	                #sFB_MCOConveyLinxAixController210(iUDT_AixConfig := #iUDT_Configuration."210".MCO_M01,
	                                                   iUDT_AixInputsModule := #iUDT_MotorInput210,
	                                                   ix_24vOk := #ix_24vOk,
	                                                   ix_SimulationModeActive := "DB_Memory".Simulation,
	                                                   ii_MotorPositionId := 1,
	                                                   qUDT_HMIStatus => #iqUDT_WorkstationStatus."210".MCO_M01,
	                                                   iqUDT_AixOutputsModule := #qUDT_MotorOutput210,
	                                                   iqUDT_ConveyorInterface := #sUDT_Interface210,
	                                                   iqUDT_MCOStatistics := #iqUDT_WorkstationStatistics."210".MCO_M01);
	            END_REGION
	        END_REGION

	        REGION 220

	            REGION Displacement
	                #sFB_Displacement220(#sUDT_Interface220);
	            END_REGION

	            REGION MCO

	                #sFB_MCOConveyLinxAixController220(iUDT_AixConfig := #iUDT_Configuration."220".MCO_M01,
	                                                   iUDT_AixInputsModule := #iUDT_MotorInput220,
	                                                   ix_24vOk := #ix_24vOk,
	                                                   ix_SimulationModeActive := "DB_Memory".Simulation,
	                                                   ii_MotorPositionId := 1,
	                                                   qUDT_HMIStatus => #iqUDT_WorkstationStatus."220".MCO_M01,
	                                                   iqUDT_AixOutputsModule := #qUDT_MotorOutput220,
	                                                   iqUDT_ConveyorInterface := #sUDT_Interface220,
	                                                   iqUDT_MCOStatistics := #iqUDT_WorkstationStatistics."220".MCO_M01);
	            END_REGION
	        END_REGION

	        REGION 221

	            REGION Displacement
	                #sFB_Displacement221(#sUDT_Interface221);
	            END_REGION

	            REGION RAT


	                #sFB_RightAngledTransfer221(iUDT_Configuration := #iUDT_Configuration."221".RightAngledTransfer,
	                                            iUDT_LowerConveyorConfiguration := #iUDT_Configuration."220".Conveyor,
	                                            iUDT_UpperConveyorConfiguration := #iUDT_Configuration."221".Conveyor,
	                                            iUDT_PECConfiguration := #iUDT_Configuration."220".PEC_EoS,
	                                            ii_DestinationA := 0,
	                                            ii_DestinationB := 0,
	                                            ii_DestinationC := 1,
	                                            ii_DestinationD := 0,
	                                            ix_HardwareOk := #ix_HardwareOk,
	                                            ix_400vOk := #ix_400vOk,
	                                            ix_24vOk := #ix_24vOk,
	                                            ix_SafetyOk := #ix_SafetyOk,
	                                            ix_AirPressureOk := #ix_AirPressureOk,
	                                            ix_SectionIsDown := #ix_SectionIsDown221,
	                                            ix_SectionIsUp := #ix_SectionIsUp221,
	                                            ix_ConveyorAAuto := FALSE,
	                                            ix_ConveyorBAuto := #iqUDT_WorkstationCommonStatus."230".AutoON,
	                                            ix_ConveyorCAuto := #iqUDT_WorkstationCommonStatus."210".AutoON,
	                                            ix_ConveyorDAuto := false,
	                                            ix_PEC := #iUDT_MotorInput220.AllSensorPortInputs.LeftSensor,
	                                            ix_ExternalReceiveRequestA := FALSE,
	                                            ix_ExternalReceiveRequestB := FALSE,
	                                            ix_ExternalReceiveRequestC := NOT #iqUDT_WorkstationStatus."210".PEC_EoS.PEC,
	                                            ix_ExternalReceiveRequestD := FALSE,
	                                            ix_PECInfeedC := #iqUDT_WorkstationStatus."210".PEC_EoS.PEC,
	                                            qUDT_HMIRATStatus => #iqUDT_WorkstationStatus."221".RightAngledTransfer,
	                                            qUDT_HMIConveyorStatus => #iqUDT_WorkstationStatus."220".Conveyor,
	                                            qUDT_HMIPECStatus => #iqUDT_WorkstationStatus."221".PEC_EoS,
	                                            qUDT_RATStatus => #iqUDT_WorkstationCommonStatus."221",
	                                            qUDT_ConveyorStatus => #iqUDT_WorkstationCommonStatus."220",
	                                            qx_PopupControl => #qx_PopupControl221,
	                                            qx_ExternalSendRequestA => #tx_dummy,
	                                            qx_ExternalSendRequestB => #tx_dummy,
	                                            qx_ExternalSendRequestC => #tx_dummy,
	                                            qx_ExternalSendRequestD => #tx_dummy,
	                                            iqUDT_EquipmentControl := #iqUDT_EquipmentControl,
	                                            iqUDT_RATCommand := #iqUDT_WorkstationCommands."221".RightAngledTransfer,
	                                            iqUDT_ConveyorCommand := #iqUDT_WorkstationCommands."220".Conveyor,
	                                            iqUDT_RATStatistics := #iqUDT_WorkstationStatistics."221".RightAngledTransfer,
	                                            iqUDT_ConveyorStatistics := #iqUDT_WorkstationStatistics."220".Conveyor,
	                                            iqUDT_PECStatistics := #iqUDT_WorkstationStatistics."221".PEC_EoS,
	                                            iqUDT_HandShakeConveyorA := #tUDT_dummyHandshake,
	                                            iqUDT_HandShakeConveyorB := #sUDT_Handshake220,
	                                            iqUDT_HandShakeConveyorC := #sUDT_Handshake210,
	                                            iqUDT_HandShakeConveyorD := #tUDT_dummyHandshake,
	                                            iqUDT_LowerConveyorInterface := #sUDT_Interface220,
	                                            iqUDT_UpperConveyorInterface := #sUDT_Interface221,
	                                            iqUDT_RATPositioning := #iqUDT_RATPositioning220,
	                                            iqUDT_BladeStopEoSInterface := #tUDT_DummyBladeStop,
	                                            iqUDT_BladeStopBoSInterface := #tUDT_DummyBladeStop);


	            END_REGION

	            REGION MCO

	                #sFB_MCOConveyLinxAixController221(iUDT_AixConfig := #iUDT_Configuration."221".MCO_M01,
	                                                   iUDT_AixInputsModule := #iUDT_MotorInput220,
	                                                   ii_PositionSetpoint := #iqUDT_RATPositioning220.Upper.EndPosition,
	                                                   ix_24vOk := #ix_24vOk,
	                                                   ix_SimulationModeActive := "DB_Memory".Simulation,
	                                                   ii_MotorPositionId := 2,
	                                                   ix_StartPositioning := #iqUDT_RATPositioning220.Upper.Start,
	                                                   ix_ResetPosition := #iqUDT_RATPositioning220.Upper.ResetPosition,
	                                                   qUDT_HMIStatus => #iqUDT_WorkstationStatus."221".MCO_M01,
	                                                   qx_Positioned => #iqUDT_RATPositioning220.Upper.Done,
	                                                   iqUDT_AixOutputsModule := #qUDT_MotorOutput220,
	                                                   iqUDT_ConveyorInterface := #sUDT_Interface221,
	                                                   iqUDT_MCOStatistics := #iqUDT_WorkstationStatistics."221".MCO_M01);
	            END_REGION

	        END_REGION

	        REGION 230

	            REGION Displacement
	                #sFB_Displacement230(#sUDT_Interface230);
	            END_REGION

	            REGION Conveyor

	                #sFB_Conveyor230(iUDT_ConveyorConfiguration := #iUDT_Configuration."230".Conveyor,
	                                 idi_PECEoSDistance := 0,
	                                 idi_PECBoSDistance := 0,
	                                 ii_ExternalSpeed := 0,
	                                 ix_SafetyOk := #ix_SafetyOk,
	                                 ix_24vOk := #ix_24vOk,
	                                 ix_400vOk := #ix_400vOk,
	                                 ix_HardwareOk := #ix_HardwareOk,
	                                 ix_PECEoS := TRUE,
	                                 ix_PECBoS := TRUE,
	                                 ix_ReverseDirection := FALSE,
	                                 ix_ExternalRequestDieBack := FALSE,
	                                 ix_ExternalRequestHold := FALSE,
	                                 ix_ResetEnergySave := FALSE,
	                                 qUDT_HMIStatus => #iqUDT_WorkstationStatus."230".Conveyor,
	                                 qUDT_Status => #iqUDT_WorkstationCommonStatus."230",
	                                 iqUDT_EquipmentControl := #iqUDT_EquipmentControl,
	                                 iqUDT_ConveyorCommand := #iqUDT_WorkstationCommands."230".Conveyor,
	                                 iqUDT_ConveyorInterface := #sUDT_Interface230,
	                                 iqUDT_HandShakeUp := #sUDT_Handshake220,
	                                 iqUDT_HandShake := #sUDT_Handshake230,
	                                 iqUDT_Statistics := #iqUDT_WorkstationStatistics."230".Conveyor);

	            END_REGION

	            REGION MCO

	                #sFB_MCOConveyLinxAixController230(iUDT_AixConfig := #iUDT_Configuration."230".MCO_M01,
	                                                   iUDT_AixInputsModule := #iUDT_MotorInput230,
	                                                   ix_24vOk := #ix_24vOk,
	                                                   ix_SimulationModeActive := "DB_Memory".Simulation,
	                                                   ii_MotorPositionId := 1,
	                                                   qUDT_HMIStatus => #iqUDT_WorkstationStatus."230".MCO_M01,
	                                                   iqUDT_AixOutputsModule := #qUDT_MotorOutput230,
	                                                   iqUDT_ConveyorInterface := #sUDT_Interface230,
	                                                   iqUDT_MCOStatistics := #iqUDT_WorkstationStatistics."230".MCO_M01);
	            END_REGION
	        END_REGION

	        REGION 240

	            REGION Displacement
	                #sFB_Displacement240(#sUDT_Interface240);
	            END_REGION

	            REGION EoS

	                #sFB_PEC240(ix_PEC := #iUDT_MotorInput240.AllSensorPortInputs.LeftSensor,
	                            iUDT_PECConfiguration := #iUDT_Configuration."240".PEC_EoS,
	                            qUDT_HMIStatus => #iqUDT_WorkstationStatus."240".PEC_EoS,
	                            iqUDT_ConveyorInterface := #sUDT_Interface240,
	                            iqUDT_PECStatistics := #iqUDT_WorkstationStatistics."240".PEC_EoS);

	            END_REGION
	            REGION Conveyor

	                #sFB_Conveyor240(iUDT_ConveyorConfiguration := #iUDT_Configuration."240".Conveyor,
	                                 idi_PECEoSDistance := #iUDT_Configuration."240".PEC_EoS.Distance,
	                                 idi_PECBoSDistance := 0,
	                                 ii_ExternalSpeed := 0,
	                                 ix_SafetyOk := #ix_SafetyOk,
	                                 ix_24vOk := #ix_24vOk,
	                                 ix_400vOk := #ix_400vOk,
	                                 ix_HardwareOk := #ix_HardwareOk,
	                                 ix_PECEoS := #iqUDT_WorkstationStatus."240".PEC_EoS.PEC,
	                                 ix_PECBoS := TRUE,
	                                 ix_ReverseDirection := FALSE,
	                                 ix_ExternalRequestDieBack := FALSE,
	                                 ix_ExternalRequestHold := FALSE,
	                                 ix_ResetEnergySave := FALSE,
	                                 qUDT_HMIStatus => #iqUDT_WorkstationStatus."240".Conveyor,
	                                 qUDT_Status => #iqUDT_WorkstationCommonStatus."240",
	                                 iqUDT_EquipmentControl := #iqUDT_EquipmentControl,
	                                 iqUDT_ConveyorCommand := #iqUDT_WorkstationCommands."240".Conveyor,
	                                 iqUDT_ConveyorInterface := #sUDT_Interface240,
	                                 iqUDT_HandShakeUp := #sUDT_Handshake230,
	                                 iqUDT_HandShake := #"sUDT_Handshake240",
	                                 iqUDT_Statistics := #iqUDT_WorkstationStatistics."240".Conveyor);

	            END_REGION

	            REGION MCO

	                #sFB_MCOConveyLinxAixController240(iUDT_AixConfig := #iUDT_Configuration."240".MCO_M01,
	                                                   iUDT_AixInputsModule := #iUDT_MotorInput240,
	                                                   ix_24vOk := #ix_24vOk,
	                                                   ix_SimulationModeActive := "DB_Memory".Simulation,
	                                                   ii_MotorPositionId := 1,
	                                                   qUDT_HMIStatus => #iqUDT_WorkstationStatus."240".MCO_M01,
	                                                   iqUDT_AixOutputsModule := #qUDT_MotorOutput240,
	                                                   iqUDT_ConveyorInterface := #sUDT_Interface240,
	                                                   iqUDT_MCOStatistics := #iqUDT_WorkstationStatistics."240".MCO_M01);
	            END_REGION

	        END_REGION

	        REGION 250

	            REGION Displacement
	                #sFB_Displacement250(#sUDT_Interface250);
	            END_REGION

	            REGION EoS

	                #sFB_PEC250(ix_PEC := #iUDT_MotorInput250.AllSensorPortInputs.LeftSensor,
	                            iUDT_PECConfiguration := #iUDT_Configuration."250".PEC_EoS,
	                            qUDT_HMIStatus => #iqUDT_WorkstationStatus."250".PEC_EoS,
	                            iqUDT_ConveyorInterface := #sUDT_Interface250,
	                            iqUDT_PECStatistics := #iqUDT_WorkstationStatistics."250".PEC_EoS);

	            END_REGION
	            REGION Conveyor

	                #sFB_Conveyor250(iUDT_ConveyorConfiguration := #iUDT_Configuration."250".Conveyor,
	                                 idi_PECEoSDistance := #iUDT_Configuration."250".PEC_EoS.Distance,
	                                 idi_PECBoSDistance := 0,
	                                 ii_ExternalSpeed := 0,
	                                 ix_SafetyOk := #ix_SafetyOk,
	                                 ix_24vOk := #ix_24vOk,
	                                 ix_400vOk := #ix_400vOk,
	                                 ix_HardwareOk := #ix_HardwareOk,
	                                 ix_PECEoS := #iqUDT_WorkstationStatus."250".PEC_EoS.PEC,
	                                 ix_PECBoS := TRUE,
	                                 ix_ReverseDirection := FALSE,
	                                 ix_ExternalRequestDieBack := FALSE,
	                                 ix_ExternalRequestHold := FALSE,
	                                 ix_ResetEnergySave := FALSE,
	                                 qUDT_HMIStatus => #iqUDT_WorkstationStatus."250".Conveyor,
	                                 qUDT_Status => #iqUDT_WorkstationCommonStatus."250",
	                                 iqUDT_EquipmentControl := #iqUDT_EquipmentControl,
	                                 iqUDT_ConveyorCommand := #iqUDT_WorkstationCommands."250".Conveyor,
	                                 iqUDT_ConveyorInterface := #sUDT_Interface250,
	                                 iqUDT_HandShakeUp := #"sUDT_Handshake240",
	                                 iqUDT_HandShake := #sUDT_Handshake250,
	                                 iqUDT_Statistics := #iqUDT_WorkstationStatistics."250".Conveyor);

	            END_REGION
	            REGION MCO

	                #sFB_MCOConveyLinxAixController250(iUDT_AixConfig := #iUDT_Configuration."250".MCO_M01,
	                                                   iUDT_AixInputsModule := #iUDT_MotorInput250,
	                                                   ix_24vOk := #ix_24vOk,
	                                                   ix_SimulationModeActive := "DB_Memory".Simulation,
	                                                   ii_MotorPositionId := 1,
	                                                   qUDT_HMIStatus => #iqUDT_WorkstationStatus."250".MCO_M01,
	                                                   iqUDT_AixOutputsModule := #qUDT_MotorOutput250,
	                                                   iqUDT_ConveyorInterface := #sUDT_Interface250,
	                                                   iqUDT_MCOStatistics := #iqUDT_WorkstationStatistics."250".MCO_M01);
	            END_REGION
	        END_REGION

	        REGION 260

	            REGION Displacement
	                #sFB_Displacement260(#sUDT_Interface260);
	            END_REGION

	            REGION EoS

	                #sFB_PEC260(ix_PEC := #iUDT_MotorInput260.AllSensorPortInputs.LeftSensor,
	                            iUDT_PECConfiguration := #iUDT_Configuration."260".PEC_EoS,
	                            qUDT_HMIStatus => #iqUDT_WorkstationStatus."260".PEC_EoS,
	                            iqUDT_ConveyorInterface := #sUDT_Interface260,
	                            iqUDT_PECStatistics := #iqUDT_WorkstationStatistics."260".PEC_EoS);

	            END_REGION
	            REGION Conveyor

	                #sFB_Conveyor260(iUDT_ConveyorConfiguration := #iUDT_Configuration."260".Conveyor,
	                                 idi_PECEoSDistance := #iUDT_Configuration."260".PEC_EoS.Distance,
	                                 idi_PECBoSDistance := 0,
	                                 ii_ExternalSpeed := 0,
	                                 ix_SafetyOk := #ix_SafetyOk,
	                                 ix_24vOk := #ix_24vOk,
	                                 ix_400vOk := #ix_400vOk,
	                                 ix_HardwareOk := #ix_HardwareOk,
	                                 ix_PECEoS := #iqUDT_WorkstationStatus."260".PEC_EoS.PEC,
	                                 ix_PECBoS := TRUE,
	                                 ix_ReverseDirection := FALSE,
	                                 ix_ExternalRequestDieBack := FALSE,
	                                 ix_ExternalRequestHold := FALSE,
	                                 ix_ResetEnergySave := FALSE,
	                                 qUDT_HMIStatus => #iqUDT_WorkstationStatus."260".Conveyor,
	                                 qUDT_Status => #iqUDT_WorkstationCommonStatus."260",
	                                 iqUDT_EquipmentControl := #iqUDT_EquipmentControl,
	                                 iqUDT_ConveyorCommand := #iqUDT_WorkstationCommands."260".Conveyor,
	                                 iqUDT_ConveyorInterface := #sUDT_Interface260,
	                                 iqUDT_HandShakeUp := #sUDT_Handshake250,
	                                 iqUDT_HandShake := #sUDT_Handshake260,
	                                 iqUDT_Statistics := #iqUDT_WorkstationStatistics."260".Conveyor);

	            END_REGION

	            REGION MCO

	                #sFB_MCOConveyLinxAixController260(iUDT_AixConfig := #iUDT_Configuration."260".MCO_M01,
	                                                   iUDT_AixInputsModule := #iUDT_MotorInput260,
	                                                   ix_24vOk := #ix_24vOk,
	                                                   ix_SimulationModeActive := "DB_Memory".Simulation,
	                                                   ii_MotorPositionId := 1,
	                                                   qUDT_HMIStatus => #iqUDT_WorkstationStatus."260".MCO_M01,
	                                                   iqUDT_AixOutputsModule := #qUDT_MotorOutput260,
	                                                   iqUDT_ConveyorInterface := #sUDT_Interface260,
	                                                   iqUDT_MCOStatistics := #iqUDT_WorkstationStatistics."260".MCO_M01);
	            END_REGION
	        END_REGION

	        REGION 270

	            REGION Displacement
	                #sFB_Displacement270(#sUDT_Interface270);
	            END_REGION

	            REGION Conveyor

	                #sFB_Conveyor270(iUDT_ConveyorConfiguration := #iUDT_Configuration."270".Conveyor,
	                                 idi_PECEoSDistance := 0,
	                                 idi_PECBoSDistance := 0,
	                                 ii_ExternalSpeed := 0,
	                                 ix_SafetyOk := #ix_SafetyOk,
	                                 ix_24vOk := #ix_24vOk,
	                                 ix_400vOk := #ix_400vOk,
	                                 ix_HardwareOk := #ix_HardwareOk,
	                                 ix_PECEoS := TRUE,
	                                 ix_PECBoS := TRUE,
	                                 ix_ReverseDirection := FALSE,
	                                 ix_ExternalRequestDieBack := FALSE,
	                                 ix_ExternalRequestHold := FALSE,
	                                 ix_ResetEnergySave := FALSE,
	                                 qUDT_HMIStatus => #iqUDT_WorkstationStatus."270".Conveyor,
	                                 qUDT_Status => #iqUDT_WorkstationCommonStatus."270",
	                                 iqUDT_EquipmentControl := #iqUDT_EquipmentControl,
	                                 iqUDT_ConveyorCommand := #iqUDT_WorkstationCommands."270".Conveyor,
	                                 iqUDT_ConveyorInterface := #sUDT_Interface270,
	                                 iqUDT_HandShakeUp := #sUDT_Handshake260,
	                                 iqUDT_HandShake := #sUDT_Handshake270,
	                                 iqUDT_Statistics := #iqUDT_WorkstationStatistics."270".Conveyor);

	            END_REGION

	            REGION MCO

	                #sFB_MCOConveyLinxAixController270(iUDT_AixConfig := #iUDT_Configuration."270".MCO_M01,
	                                                   iUDT_AixInputsModule := #iUDT_MotorInput270,
	                                                   ix_24vOk := #ix_24vOk,
	                                                   ix_SimulationModeActive := "DB_Memory".Simulation,
	                                                   ii_MotorPositionId := 1,
	                                                   qUDT_HMIStatus => #iqUDT_WorkstationStatus."270".MCO_M01,
	                                                   iqUDT_AixOutputsModule := #qUDT_MotorOutput270,
	                                                   iqUDT_ConveyorInterface := #sUDT_Interface270,
	                                                   iqUDT_MCOStatistics := #iqUDT_WorkstationStatistics."270".MCO_M01);
	            END_REGION
	        END_REGION

	        REGION 280

	            REGION Displacement
	                #sFB_Displacement280(#sUDT_Interface280);
	            END_REGION

	            REGION EoS

	                #sFB_PEC280(ix_PEC := #iUDT_MotorInput280.AllSensorPortInputs.LeftSensor,
	                            iUDT_PECConfiguration := #iUDT_Configuration."280".PEC_EoS,
	                            qUDT_HMIStatus => #iqUDT_WorkstationStatus."280".PEC_EoS,
	                            iqUDT_ConveyorInterface := #sUDT_Interface280,
	                            iqUDT_PECStatistics := #iqUDT_WorkstationStatistics."280".PEC_EoS);

	            END_REGION

	            REGION Scanner

	                #sFB_CognexDM280(iUDT_CognexDM260_IN := #iUDT_ScannerInput280,
	                                 iqUDT_EquipmentControl := #iqUDT_EquipmentControl,
	                                 ix_Trigger := NOT #iqUDT_WorkstationStatus."280".PEC_EoS.PEC,
	                                 qUDT_CognexDM260_OUT => #qUDT_ScannerOutput280,
	                                 qs_Barcode => #ss_Barcode280,
	                                 qw_RetVal => #tw_dummy);

	            END_REGION

	            REGION Conveyor

	                #sUDT_Handshake280.RTR := #sUDT_Handshake280.RTR OR #iqUDT_WorkstationStatus."280".PEC_EoS.PEC;

	                #sFB_Conveyor280(iUDT_ConveyorConfiguration := #iUDT_Configuration."280".Conveyor,
	                                 idi_PECEoSDistance := #iUDT_Configuration."280".PEC_EoS.Distance,
	                                 idi_PECBoSDistance := 0,
	                                 ii_ExternalSpeed := 0,
	                                 ix_SafetyOk := #ix_SafetyOk,
	                                 ix_24vOk := #ix_24vOk,
	                                 ix_400vOk := #ix_400vOk,
	                                 ix_HardwareOk := #ix_HardwareOk,
	                                 ix_PECEoS := #iqUDT_WorkstationStatus."280".PEC_EoS.PEC,
	                                 ix_PECBoS := TRUE,
	                                 ix_ReverseDirection := FALSE,
	                                 ix_ExternalRequestDieBack := FALSE,
	                                 ix_ExternalRequestHold := FALSE,
	                                 ix_ResetEnergySave := FALSE,
	                                 qUDT_HMIStatus => #iqUDT_WorkstationStatus."280".Conveyor,
	                                 qUDT_Status => #iqUDT_WorkstationCommonStatus."280",
	                                 iqUDT_EquipmentControl := #iqUDT_EquipmentControl,
	                                 iqUDT_ConveyorCommand := #iqUDT_WorkstationCommands."280".Conveyor,
	                                 iqUDT_ConveyorInterface := #sUDT_Interface280,
	                                 iqUDT_HandShakeUp := #sUDT_Handshake270,
	                                 iqUDT_HandShake := #sUDT_Handshake280,
	                                 iqUDT_Statistics := #iqUDT_WorkstationStatistics."280".Conveyor);

	            END_REGION

	            REGION MCO

	                #sFB_MCOConveyLinxAixController280(iUDT_AixConfig := #iUDT_Configuration."280".MCO_M01,
	                                                   iUDT_AixInputsModule := #iUDT_MotorInput280,
	                                                   ix_24vOk := #ix_24vOk,
	                                                   ix_SimulationModeActive := "DB_Memory".Simulation,
	                                                   ii_MotorPositionId := 1,
	                                                   qUDT_HMIStatus => #iqUDT_WorkstationStatus."280".MCO_M01,
	                                                   iqUDT_AixOutputsModule := #qUDT_MotorOutput280,
	                                                   iqUDT_ConveyorInterface := #sUDT_Interface280,
	                                                   iqUDT_MCOStatistics := #iqUDT_WorkstationStatistics."280".MCO_M01);
	            END_REGION
	        END_REGION


	        REGION 290

	            REGION Displacement
	                #sFB_Displacement290(#sUDT_Interface290);
	            END_REGION

	            REGION MCO

	                #sFB_MCOConveyLinxAixController290(iUDT_AixConfig := #iUDT_Configuration."290".MCO_M01,
	                                                   iUDT_AixInputsModule := #iUDT_MotorInput290,
	                                                   ii_PositionSetpoint := #iqUDT_RATPositioning290.Lower.EndPosition,
	                                                   ix_24vOk := #ix_24vOk,
	                                                   ix_SimulationModeActive := "DB_Memory".Simulation,
	                                                   ii_MotorPositionId := 1,
	                                                   ix_StartPositioning := #iqUDT_RATPositioning290.Lower.Start,
	                                                   ix_ResetPosition := #iqUDT_RATPositioning290.Lower.ResetPosition,
	                                                   qUDT_HMIStatus => #iqUDT_WorkstationStatus."290".MCO_M01,
	                                                   qx_Positioned => #iqUDT_RATPositioning290.Lower.Done,
	                                                   iqUDT_AixOutputsModule := #qUDT_MotorOutput290,
	                                                   iqUDT_ConveyorInterface := #sUDT_Interface290,
	                                                   iqUDT_MCOStatistics := #iqUDT_WorkstationStatistics."290".MCO_M01);
	            END_REGION
	        END_REGION

	        REGION 291

	            REGION Displacement
	                #sFB_Displacement291(#sUDT_Interface291);
	            END_REGION

	            REGION RAT

	                #sFB_RightAngledTransfer291(iUDT_Configuration := #iUDT_Configuration."291".RightAngledTransfer,
	                                            iUDT_LowerConveyorConfiguration := #iUDT_Configuration."290".Conveyor,
	                                            iUDT_UpperConveyorConfiguration := #iUDT_Configuration."291".Conveyor,
	                                            iUDT_PECConfiguration := #iUDT_Configuration."290".PEC_EoS,
	                                            ii_DestinationA := #si_DestinationA291,
	                                            ii_DestinationB := 0,
	                                            ii_DestinationC := 0,
	                                            ii_DestinationD := 0,
	                                            ix_HardwareOk := #ix_HardwareOk,
	                                            ix_400vOk := #ix_400vOk,
	                                            ix_24vOk := #ix_24vOk,
	                                            ix_SafetyOk := #ix_SafetyOk,
	                                            ix_AirPressureOk := #ix_AirPressureOk,
	                                            ix_SectionIsDown := #ix_SectionIsDown291,
	                                            ix_SectionIsUp := #ix_SectionIsUp291,
	                                            ix_ConveyorAAuto := #iqUDT_WorkstationCommonStatus."280".AutoON,
	                                            ix_ConveyorBAuto := FALSE,
	                                            ix_ConveyorCAuto := #iqUDT_WorkstationCommonStatus."300".AutoON,
	                                            ix_ConveyorDAuto := FALSE,
	                                            ix_PEC := #iUDT_MotorInput290.AllSensorPortInputs.LeftSensor,
	                                            ix_ExternalReceiveRequestA := NOT #iqUDT_WorkstationStatus."280".PEC_EoS.PEC,
	                                            ix_ExternalReceiveRequestB := FALSE,
	                                            ix_ExternalReceiveRequestC := FALSE,
	                                            ix_ExternalReceiveRequestD := FALSE,
	                                            ix_PECInfeedA := #iqUDT_WorkstationStatus."280".PEC_EoS.PEC,
	                                            qUDT_HMIRATStatus => #iqUDT_WorkstationStatus."291".RightAngledTransfer,
	                                            qUDT_HMIConveyorStatus => #iqUDT_WorkstationStatus."290".Conveyor,
	                                            qUDT_HMIPECStatus => #iqUDT_WorkstationStatus."291".PEC_EoS,
	                                            qUDT_RATStatus => #iqUDT_WorkstationCommonStatus."291",
	                                            qUDT_ConveyorStatus => #iqUDT_WorkstationCommonStatus."290",
	                                            qx_PopupControl => #qx_PopupControl291,
	                                            qx_ExternalSendRequestA => #tx_dummy,
	                                            qx_ExternalSendRequestB => #tx_dummy,
	                                            qx_ExternalSendRequestC => #tx_dummy,
	                                            qx_ExternalSendRequestD => #tx_dummy,
	                                            iqUDT_EquipmentControl := #iqUDT_EquipmentControl,
	                                            iqUDT_RATCommand := #iqUDT_WorkstationCommands."291".RightAngledTransfer,
	                                            iqUDT_ConveyorCommand := #iqUDT_WorkstationCommands."290".Conveyor,
	                                            iqUDT_RATStatistics := #iqUDT_WorkstationStatistics."291".RightAngledTransfer,
	                                            iqUDT_ConveyorStatistics := #iqUDT_WorkstationStatistics."290".Conveyor,
	                                            iqUDT_PECStatistics := #iqUDT_WorkstationStatistics."291".PEC_EoS,
	                                            iqUDT_HandShakeConveyorA := #sUDT_Handshake280,
	                                            iqUDT_HandShakeConveyorB := #tUDT_dummyHandshake,
	                                            iqUDT_HandShakeConveyorC := #sUDT_HandshakeUp291,
	                                            iqUDT_HandShakeConveyorD := #tUDT_dummyHandshake,
	                                            iqUDT_LowerConveyorInterface := #sUDT_Interface290,
	                                            iqUDT_UpperConveyorInterface := #sUDT_Interface291,
	                                            iqUDT_RATPositioning := #iqUDT_RATPositioning290,
	                                            iqUDT_BladeStopEoSInterface := #tUDT_DummyBladeStop,
	                                            iqUDT_BladeStopBoSInterface := #tUDT_DummyBladeStop);

	            END_REGION

	            REGION MCO

	                #sFB_MCOConveyLinxAixController291(iUDT_AixConfig := #iUDT_Configuration."291".MCO_M01,
	                                                   iUDT_AixInputsModule := #iUDT_MotorInput290,
	                                                   ix_24vOk := #ix_24vOk,
	                                                   ix_SimulationModeActive := "DB_Memory".Simulation,
	                                                   ii_MotorPositionId := 2,
	                                                   qUDT_HMIStatus => #iqUDT_WorkstationStatus."291".MCO_M01,
	                                                   iqUDT_AixOutputsModule := #qUDT_MotorOutput290,
	                                                   iqUDT_ConveyorInterface := #sUDT_Interface291,
	                                                   iqUDT_MCOStatistics := #iqUDT_WorkstationStatistics."290".MCO_M01);
	            END_REGION

	        END_REGION

	        REGION 300

	            REGION Displacement
	                #sFB_Displacement300(#sUDT_Interface300);
	            END_REGION

	            REGION EoS

	                #sFB_PEC300(ix_PEC := #iUDT_MotorInput300.AllSensorPortInputs.LeftSensor,
	                            iUDT_PECConfiguration := #iUDT_Configuration."300".PEC_EoS,
	                            qUDT_HMIStatus => #iqUDT_WorkstationStatus."300".PEC_EoS,
	                            iqUDT_ConveyorInterface := #sUDT_Interface300,
	                            iqUDT_PECStatistics := #iqUDT_WorkstationStatistics."300".PEC_EoS);

	            END_REGION
	            REGION Conveyor

	                #sUDT_Handshake300.RTR := #sUDT_Handshake300.RTR OR #iqUDT_WorkstationStatus."300".PEC_EoS.PEC;

	                #sFB_Conveyor300(iUDT_ConveyorConfiguration := #iUDT_Configuration."300".Conveyor,
	                                 idi_PECEoSDistance := #iUDT_Configuration."300".PEC_EoS.Distance,
	                                 idi_PECBoSDistance := 0,
	                                 ii_ExternalSpeed := 0,
	                                 ix_SafetyOk := #ix_SafetyOk,
	                                 ix_24vOk := #ix_24vOk,
	                                 ix_400vOk := #ix_400vOk,
	                                 ix_HardwareOk := #ix_HardwareOk,
	                                 ix_PECEoS := #iqUDT_WorkstationStatus."300".PEC_EoS.PEC,
	                                 ix_PECBoS := TRUE,
	                                 ix_ReverseDirection := FALSE,
	                                 ix_ExternalRequestDieBack := FALSE,
	                                 ix_ExternalRequestHold := FALSE,
	                                 ix_ResetEnergySave := FALSE,
	                                 qUDT_HMIStatus => #iqUDT_WorkstationStatus."300".Conveyor,
	                                 qUDT_Status => #iqUDT_WorkstationCommonStatus."300",
	                                 iqUDT_EquipmentControl := #iqUDT_EquipmentControl,
	                                 iqUDT_ConveyorCommand := #iqUDT_WorkstationCommands."300".Conveyor,
	                                 iqUDT_ConveyorInterface := #sUDT_Interface300,
	                                 iqUDT_HandShakeUp := #sUDT_HandshakeUp291,
	                                 iqUDT_HandShake := #sUDT_Handshake300,
	                                 iqUDT_Statistics := #iqUDT_WorkstationStatistics."300".Conveyor);

	            END_REGION
	            REGION MCO

	                #sFB_MCOConveyLinxAixController300(iUDT_AixConfig := #iUDT_Configuration."300".MCO_M01,
	                                                   iUDT_AixInputsModule := #iUDT_MotorInput300,
	                                                   ix_24vOk := #ix_24vOk,
	                                                   ix_SimulationModeActive := "DB_Memory".Simulation,
	                                                   ii_MotorPositionId := 1,
	                                                   qUDT_HMIStatus => #iqUDT_WorkstationStatus."300".MCO_M01,
	                                                   iqUDT_AixOutputsModule := #qUDT_MotorOutput300,
	                                                   iqUDT_ConveyorInterface := #sUDT_Interface300,
	                                                   iqUDT_MCOStatistics := #iqUDT_WorkstationStatistics."300".MCO_M01);
	            END_REGION
	        END_REGION
	    END_IF;
	END_REGION

	REGION 5 - Left Station
	    IF #iUDT_Configuration.GlobalConfig.LeftStationExists THEN
	        REGION 410

	            REGION Displacement
	                #sFB_Displacement410(#sUDT_Interface410);
	            END_REGION

	            REGION EoS

	                #sFB_PEC410(ix_PEC := #iUDT_MotorInput410.AllSensorPortInputs.LeftSensor,
	                            iUDT_PECConfiguration := #iUDT_Configuration."410".PEC_EoS,
	                            qUDT_HMIStatus => #iqUDT_WorkstationStatus."410".PEC_EoS,
	                            iqUDT_ConveyorInterface := #sUDT_Interface410,
	                            iqUDT_PECStatistics := #iqUDT_WorkstationStatistics."410".PEC_EoS);

	            END_REGION
	            REGION Conveyor

	                #sUDT_Handshake410.RTR := #sUDT_Handshake410.RTR OR #iqUDT_WorkstationStatus."410".PEC_EoS.PEC;

	                #sFB_Conveyor410(iUDT_ConveyorConfiguration := #iUDT_Configuration."410".Conveyor,
	                                 idi_PECEoSDistance := #iUDT_Configuration."410".PEC_EoS.Distance,
	                                 idi_PECBoSDistance := 0,
	                                 ii_ExternalSpeed := 0,
	                                 ix_SafetyOk := #ix_SafetyOk,
	                                 ix_24vOk := #ix_24vOk,
	                                 ix_400vOk := #ix_400vOk,
	                                 ix_HardwareOk := #ix_HardwareOk,
	                                 ix_PECEoS := #iqUDT_WorkstationStatus."410".PEC_EoS.PEC,
	                                 ix_PECBoS := TRUE,
	                                 ix_ReverseDirection := FALSE,
	                                 ix_ExternalRequestDieBack := FALSE,
	                                 ix_ExternalRequestHold := FALSE,
	                                 ix_ResetEnergySave := FALSE,
	                                 qUDT_HMIStatus => #iqUDT_WorkstationStatus."410".Conveyor,
	                                 qUDT_Status => #iqUDT_WorkstationCommonStatus."410",
	                                 iqUDT_EquipmentControl := #iqUDT_EquipmentControl,
	                                 iqUDT_ConveyorCommand := #iqUDT_WorkstationCommands."410".Conveyor,
	                                 iqUDT_ConveyorInterface := #sUDT_Interface410,
	                                 iqUDT_HandShakeUp := #sUDT_Handshake121,
	                                 iqUDT_HandShake := #sUDT_Handshake410,
	                                 iqUDT_Statistics := #iqUDT_WorkstationStatistics."410".Conveyor);

	            END_REGION
	            REGION MCO

	                #sFB_MCOConveyLinxAixController410(iUDT_AixConfig := #iUDT_Configuration."410".MCO_M01,
	                                                   iUDT_AixInputsModule := #iUDT_MotorInput410,
	                                                   ix_24vOk := #ix_24vOk,
	                                                   ix_SimulationModeActive := "DB_Memory".Simulation,
	                                                   ii_MotorPositionId := 1,
	                                                   qUDT_HMIStatus => #iqUDT_WorkstationStatus."410".MCO_M01,
	                                                   iqUDT_AixOutputsModule := #qUDT_MotorOutput410,
	                                                   iqUDT_ConveyorInterface := #sUDT_Interface410,
	                                                   iqUDT_MCOStatistics := #iqUDT_WorkstationStatistics."410".MCO_M01);
	            END_REGION
	        END_REGION

	        REGION 420

	            REGION Displacement
	                #sFB_Displacement420(#sUDT_Interface420);
	            END_REGION

	            REGION MCO

	                #sFB_MCOConveyLinxAixController420(iUDT_AixConfig := #iUDT_Configuration."420".MCO_M01,
	                                                   iUDT_AixInputsModule := #iUDT_MotorInput420,
	                                                   ix_24vOk := #ix_24vOk,
	                                                   ix_SimulationModeActive := "DB_Memory".Simulation,
	                                                   ii_MotorPositionId := 1,
	                                                   qUDT_HMIStatus => #iqUDT_WorkstationStatus."420".MCO_M01,
	                                                   iqUDT_AixOutputsModule := #qUDT_MotorOutput420,
	                                                   iqUDT_ConveyorInterface := #sUDT_Interface420,
	                                                   iqUDT_MCOStatistics := #iqUDT_WorkstationStatistics."420".MCO_M01);
	            END_REGION
	        END_REGION

	        REGION 421

	            REGION Displacement
	                #sFB_Displacement421(#sUDT_Interface421);
	            END_REGION

	            REGION RAT

	                #sFB_RightAngledTransfer421(iUDT_Configuration := #iUDT_Configuration."421".RightAngledTransfer,
	                                            iUDT_LowerConveyorConfiguration := #iUDT_Configuration."420".Conveyor,
	                                            iUDT_UpperConveyorConfiguration := #iUDT_Configuration."421".Conveyor,
	                                            iUDT_PECConfiguration := #iUDT_Configuration."420".PEC_EoS,
	                                            ii_DestinationA := 0,
	                                            ii_DestinationB := 0,
	                                            ii_DestinationC := 0,
	                                            ii_DestinationD := 1,
	                                            ix_HardwareOk := #ix_HardwareOk,
	                                            ix_400vOk := #ix_400vOk,
	                                            ix_24vOk := #ix_24vOk,
	                                            ix_SafetyOk := #ix_SafetyOk,
	                                            ix_AirPressureOk := #ix_AirPressureOk,
	                                            ix_SectionIsDown := #ix_SectionIsDown421,
	                                            ix_SectionIsUp := #ix_SectionIsUp421,
	                                            ix_ConveyorAAuto := FALSE,
	                                            ix_ConveyorBAuto := #iqUDT_WorkstationCommonStatus."430".AutoON,
	                                            ix_ConveyorCAuto := FALSE,
	                                            ix_ConveyorDAuto := #iqUDT_WorkstationCommonStatus."410".AutoON,
	                                            ix_PEC := #iUDT_MotorInput420.AllSensorPortInputs.LeftSensor,
	                                            ix_ExternalReceiveRequestA := FALSE,
	                                            ix_ExternalReceiveRequestB := FALSE,
	                                            ix_ExternalReceiveRequestC := FALSE,
	                                            ix_ExternalReceiveRequestD := NOT #iqUDT_WorkstationStatus."410".PEC_EoS.PEC,
	                                            ix_PECInfeedA := false,
	                                            ix_PECInfeedD := #iqUDT_WorkstationStatus."410".PEC_EoS.PEC,
	                                            qUDT_HMIRATStatus => #iqUDT_WorkstationStatus."421".RightAngledTransfer,
	                                            qUDT_HMIConveyorStatus => #iqUDT_WorkstationStatus."420".Conveyor,
	                                            qUDT_HMIPECStatus => #iqUDT_WorkstationStatus."421".PEC_EoS,
	                                            qUDT_RATStatus => #iqUDT_WorkstationCommonStatus."421",
	                                            qUDT_ConveyorStatus => #iqUDT_WorkstationCommonStatus."420",
	                                            qx_PopupControl => #qx_PopupControl421,
	                                            qx_ExternalSendRequestA => #tx_dummy,
	                                            qx_ExternalSendRequestB => #tx_dummy,
	                                            qx_ExternalSendRequestC => #tx_dummy,
	                                            qx_ExternalSendRequestD => #tx_dummy,
	                                            iqUDT_EquipmentControl := #iqUDT_EquipmentControl,
	                                            iqUDT_RATCommand := #iqUDT_WorkstationCommands."421".RightAngledTransfer,
	                                            iqUDT_ConveyorCommand := #iqUDT_WorkstationCommands."420".Conveyor,
	                                            iqUDT_RATStatistics := #iqUDT_WorkstationStatistics."421".RightAngledTransfer,
	                                            iqUDT_ConveyorStatistics := #iqUDT_WorkstationStatistics."420".Conveyor,
	                                            iqUDT_PECStatistics := #iqUDT_WorkstationStatistics."421".PEC_EoS,
	                                            iqUDT_HandShakeConveyorA := #tUDT_dummyHandshake,
	                                            iqUDT_HandShakeConveyorB := #sUDT_Handshake420,
	                                            iqUDT_HandShakeConveyorC := #tUDT_dummyHandshake,
	                                            iqUDT_HandShakeConveyorD := #sUDT_Handshake410,
	                                            iqUDT_LowerConveyorInterface := #sUDT_Interface420,
	                                            iqUDT_UpperConveyorInterface := #sUDT_Interface421,
	                                            iqUDT_RATPositioning := #iqUDT_RATPositioning420,
	                                            iqUDT_BladeStopEoSInterface := #tUDT_DummyBladeStop,
	                                            iqUDT_BladeStopBoSInterface := #tUDT_DummyBladeStop);

	            END_REGION

	            REGION MCO

	                #sFB_MCOConveyLinxAixController421(iUDT_AixConfig := #iUDT_Configuration."421".MCO_M01,
	                                                   iUDT_AixInputsModule := #iUDT_MotorInput420,
	                                                   ii_PositionSetpoint := #iqUDT_RATPositioning420.Upper.EndPosition,
	                                                   ix_24vOk := #ix_24vOk,
	                                                   ix_SimulationModeActive := "DB_Memory".Simulation,
	                                                   ii_MotorPositionId := 2,
	                                                   ix_StartPositioning := #iqUDT_RATPositioning420.Upper.Start,
	                                                   ix_ResetPosition := #iqUDT_RATPositioning420.Upper.ResetPosition,
	                                                   qUDT_HMIStatus => #iqUDT_WorkstationStatus."421".MCO_M01,
	                                                   qx_Positioned => #iqUDT_RATPositioning420.Upper.Done,
	                                                   iqUDT_AixOutputsModule := #qUDT_MotorOutput420,
	                                                   iqUDT_ConveyorInterface := #sUDT_Interface421,
	                                                   iqUDT_MCOStatistics := #iqUDT_WorkstationStatistics."421".MCO_M01);
	            END_REGION

	        END_REGION

	        REGION 430

	            REGION Displacement
	                #sFB_Displacement430(#sUDT_Interface430);
	            END_REGION

	            REGION Conveyor

	                #sFB_Conveyor430(iUDT_ConveyorConfiguration := #iUDT_Configuration."430".Conveyor,
	                                 idi_PECEoSDistance := 0,
	                                 idi_PECBoSDistance := 0,
	                                 ii_ExternalSpeed := 0,
	                                 ix_SafetyOk := #ix_SafetyOk,
	                                 ix_24vOk := #ix_24vOk,
	                                 ix_400vOk := #ix_400vOk,
	                                 ix_HardwareOk := #ix_HardwareOk,
	                                 ix_PECEoS := TRUE,
	                                 ix_PECBoS := TRUE,
	                                 ix_ReverseDirection := FALSE,
	                                 ix_ExternalRequestDieBack := FALSE,
	                                 ix_ExternalRequestHold := FALSE,
	                                 ix_ResetEnergySave := FALSE,
	                                 qUDT_HMIStatus => #iqUDT_WorkstationStatus."430".Conveyor,
	                                 qUDT_Status => #iqUDT_WorkstationCommonStatus."430",
	                                 iqUDT_EquipmentControl := #iqUDT_EquipmentControl,
	                                 iqUDT_ConveyorCommand := #iqUDT_WorkstationCommands."430".Conveyor,
	                                 iqUDT_ConveyorInterface := #sUDT_Interface430,
	                                 iqUDT_HandShakeUp := #sUDT_Handshake420,
	                                 iqUDT_HandShake := #sUDT_Handshake430,
	                                 iqUDT_Statistics := #iqUDT_WorkstationStatistics."430".Conveyor);

	            END_REGION
	            REGION MCO

	                #sFB_MCOConveyLinxAixController430(iUDT_AixConfig := #iUDT_Configuration."430".MCO_M01,
	                                                   iUDT_AixInputsModule := #iUDT_MotorInput430,
	                                                   ix_24vOk := #ix_24vOk,
	                                                   ix_SimulationModeActive := "DB_Memory".Simulation,
	                                                   ii_MotorPositionId := 1,
	                                                   qUDT_HMIStatus => #iqUDT_WorkstationStatus."430".MCO_M01,
	                                                   iqUDT_AixOutputsModule := #qUDT_MotorOutput430,
	                                                   iqUDT_ConveyorInterface := #sUDT_Interface430,
	                                                   iqUDT_MCOStatistics := #iqUDT_WorkstationStatistics."430".MCO_M01);
	            END_REGION
	        END_REGION

	        REGION 440

	            REGION Displacement
	                #sFB_Displacement440(#sUDT_Interface440);
	            END_REGION

	            REGION EoS

	                #sFB_PEC440(ix_PEC := #iUDT_MotorInput440.AllSensorPortInputs.LeftSensor,
	                            iUDT_PECConfiguration := #iUDT_Configuration."440".PEC_EoS,
	                            qUDT_HMIStatus => #iqUDT_WorkstationStatus."440".PEC_EoS,
	                            iqUDT_ConveyorInterface := #sUDT_Interface440,
	                            iqUDT_PECStatistics := #iqUDT_WorkstationStatistics."440".PEC_EoS);

	            END_REGION
	            REGION Conveyor

	                #sFB_Conveyor440(iUDT_ConveyorConfiguration := #iUDT_Configuration."440".Conveyor,
	                                 idi_PECEoSDistance := #iUDT_Configuration."440".PEC_EoS.Distance,
	                                 idi_PECBoSDistance := 0,
	                                 ii_ExternalSpeed := 0,
	                                 ix_SafetyOk := #ix_SafetyOk,
	                                 ix_24vOk := #ix_24vOk,
	                                 ix_400vOk := #ix_400vOk,
	                                 ix_HardwareOk := #ix_HardwareOk,
	                                 ix_PECEoS := #iqUDT_WorkstationStatus."440".PEC_EoS.PEC,
	                                 ix_PECBoS := TRUE,
	                                 ix_ReverseDirection := FALSE,
	                                 ix_ExternalRequestDieBack := FALSE,
	                                 ix_ExternalRequestHold := FALSE,
	                                 ix_ResetEnergySave := FALSE,
	                                 qUDT_HMIStatus => #iqUDT_WorkstationStatus."440".Conveyor,
	                                 qUDT_Status => #iqUDT_WorkstationCommonStatus."440",
	                                 iqUDT_EquipmentControl := #iqUDT_EquipmentControl,
	                                 iqUDT_ConveyorCommand := #iqUDT_WorkstationCommands."440".Conveyor,
	                                 iqUDT_ConveyorInterface := #sUDT_Interface440,
	                                 iqUDT_HandShakeUp := #sUDT_Handshake430,
	                                 iqUDT_HandShake := #sUDT_Handshake440,
	                                 iqUDT_Statistics := #iqUDT_WorkstationStatistics."440".Conveyor);

	            END_REGION

	            REGION MCO

	                #sFB_MCOConveyLinxAixController440(iUDT_AixConfig := #iUDT_Configuration."440".MCO_M01,
	                                                   iUDT_AixInputsModule := #iUDT_MotorInput440,
	                                                   ix_24vOk := #ix_24vOk,
	                                                   ix_SimulationModeActive := "DB_Memory".Simulation,
	                                                   ii_MotorPositionId := 1,
	                                                   qUDT_HMIStatus => #iqUDT_WorkstationStatus."440".MCO_M01,
	                                                   iqUDT_AixOutputsModule := #qUDT_MotorOutput440,
	                                                   iqUDT_ConveyorInterface := #sUDT_Interface440,
	                                                   iqUDT_MCOStatistics := #iqUDT_WorkstationStatistics."440".MCO_M01);
	            END_REGION
	        END_REGION

	        REGION 450

	            REGION Displacement
	                #sFB_Displacement450(#sUDT_Interface450);
	            END_REGION

	            REGION EoS

	                #sFB_PEC450(ix_PEC := #iUDT_MotorInput450.AllSensorPortInputs.LeftSensor,
	                            iUDT_PECConfiguration := #iUDT_Configuration."450".PEC_EoS,
	                            qUDT_HMIStatus => #iqUDT_WorkstationStatus."450".PEC_EoS,
	                            iqUDT_ConveyorInterface := #sUDT_Interface450,
	                            iqUDT_PECStatistics := #iqUDT_WorkstationStatistics."450".PEC_EoS);

	            END_REGION
	            REGION Conveyor

	                #sFB_Conveyor450(iUDT_ConveyorConfiguration := #iUDT_Configuration."450".Conveyor,
	                                 idi_PECEoSDistance := #iUDT_Configuration."450".PEC_EoS.Distance,
	                                 idi_PECBoSDistance := 0,
	                                 ii_ExternalSpeed := 0,
	                                 ix_SafetyOk := #ix_SafetyOk,
	                                 ix_24vOk := #ix_24vOk,
	                                 ix_400vOk := #ix_400vOk,
	                                 ix_HardwareOk := #ix_HardwareOk,
	                                 ix_PECEoS := #iqUDT_WorkstationStatus."450".PEC_EoS.PEC,
	                                 ix_PECBoS := TRUE,
	                                 ix_ReverseDirection := FALSE,
	                                 ix_ExternalRequestDieBack := FALSE,
	                                 ix_ExternalRequestHold := FALSE,
	                                 ix_ResetEnergySave := FALSE,
	                                 qUDT_HMIStatus => #iqUDT_WorkstationStatus."450".Conveyor,
	                                 qUDT_Status => #iqUDT_WorkstationCommonStatus."450",
	                                 iqUDT_EquipmentControl := #iqUDT_EquipmentControl,
	                                 iqUDT_ConveyorCommand := #iqUDT_WorkstationCommands."450".Conveyor,
	                                 iqUDT_ConveyorInterface := #sUDT_Interface450,
	                                 iqUDT_HandShakeUp := #sUDT_Handshake440,
	                                 iqUDT_HandShake := #sUDT_Handshake450,
	                                 iqUDT_Statistics := #iqUDT_WorkstationStatistics."450".Conveyor);

	            END_REGION
	            REGION MCO

	                #sFB_MCOConveyLinxAixController450(iUDT_AixConfig := #iUDT_Configuration."450".MCO_M01,
	                                                   iUDT_AixInputsModule := #iUDT_MotorInput450,
	                                                   ix_24vOk := #ix_24vOk,
	                                                   ix_SimulationModeActive := "DB_Memory".Simulation,
	                                                   ii_MotorPositionId := 1,
	                                                   qUDT_HMIStatus => #iqUDT_WorkstationStatus."450".MCO_M01,
	                                                   iqUDT_AixOutputsModule := #qUDT_MotorOutput450,
	                                                   iqUDT_ConveyorInterface := #sUDT_Interface450,
	                                                   iqUDT_MCOStatistics := #iqUDT_WorkstationStatistics."450".MCO_M01);
	            END_REGION
	        END_REGION

	        REGION 460

	            REGION Displacement
	                #sFB_Displacement460(#sUDT_Interface460);
	            END_REGION

	            REGION EoS

	                #sFB_PEC460(ix_PEC := #iUDT_MotorInput460.AllSensorPortInputs.LeftSensor,
	                            iUDT_PECConfiguration := #iUDT_Configuration."460".PEC_EoS,
	                            qUDT_HMIStatus => #iqUDT_WorkstationStatus."460".PEC_EoS,
	                            iqUDT_ConveyorInterface := #sUDT_Interface460,
	                            iqUDT_PECStatistics := #iqUDT_WorkstationStatistics."460".PEC_EoS);

	            END_REGION
	            REGION Conveyor

	                #sFB_Conveyor460(iUDT_ConveyorConfiguration := #iUDT_Configuration."460".Conveyor,
	                                 idi_PECEoSDistance := #iUDT_Configuration."460".PEC_EoS.Distance,
	                                 idi_PECBoSDistance := 0,
	                                 ii_ExternalSpeed := 0,
	                                 ix_SafetyOk := #ix_SafetyOk,
	                                 ix_24vOk := #ix_24vOk,
	                                 ix_400vOk := #ix_400vOk,
	                                 ix_HardwareOk := #ix_HardwareOk,
	                                 ix_PECEoS := #iqUDT_WorkstationStatus."460".PEC_EoS.PEC,
	                                 ix_PECBoS := TRUE,
	                                 ix_ReverseDirection := FALSE,
	                                 ix_ExternalRequestDieBack := FALSE,
	                                 ix_ExternalRequestHold := FALSE,
	                                 ix_ResetEnergySave := FALSE,
	                                 qUDT_HMIStatus => #iqUDT_WorkstationStatus."460".Conveyor,
	                                 qUDT_Status => #iqUDT_WorkstationCommonStatus."460",
	                                 iqUDT_EquipmentControl := #iqUDT_EquipmentControl,
	                                 iqUDT_ConveyorCommand := #iqUDT_WorkstationCommands."460".Conveyor,
	                                 iqUDT_ConveyorInterface := #sUDT_Interface460,
	                                 iqUDT_HandShakeUp := #sUDT_Handshake450,
	                                 iqUDT_HandShake := #sUDT_Handshake460,
	                                 iqUDT_Statistics := #iqUDT_WorkstationStatistics."460".Conveyor);

	            END_REGION

	            REGION MCO

	                #sFB_MCOConveyLinxAixController460(iUDT_AixConfig := #iUDT_Configuration."460".MCO_M01,
	                                                   iUDT_AixInputsModule := #iUDT_MotorInput460,
	                                                   ix_24vOk := #ix_24vOk,
	                                                   ix_SimulationModeActive := "DB_Memory".Simulation,
	                                                   ii_MotorPositionId := 1,
	                                                   qUDT_HMIStatus => #iqUDT_WorkstationStatus."460".MCO_M01,
	                                                   iqUDT_AixOutputsModule := #qUDT_MotorOutput460,
	                                                   iqUDT_ConveyorInterface := #sUDT_Interface460,
	                                                   iqUDT_MCOStatistics := #iqUDT_WorkstationStatistics."460".MCO_M01);
	            END_REGION
	        END_REGION

	        REGION 470

	            REGION Displacement
	                #sFB_Displacement470(#sUDT_Interface470);
	            END_REGION

	            REGION Conveyor

	                #sFB_Conveyor470(iUDT_ConveyorConfiguration := #iUDT_Configuration."470".Conveyor,
	                                 idi_PECEoSDistance := 0,
	                                 idi_PECBoSDistance := 0,
	                                 ii_ExternalSpeed := 0,
	                                 ix_SafetyOk := #ix_SafetyOk,
	                                 ix_24vOk := #ix_24vOk,
	                                 ix_400vOk := #ix_400vOk,
	                                 ix_HardwareOk := #ix_HardwareOk,
	                                 ix_PECEoS := TRUE,
	                                 ix_PECBoS := TRUE,
	                                 ix_ReverseDirection := FALSE,
	                                 ix_ExternalRequestDieBack := FALSE,
	                                 ix_ExternalRequestHold := FALSE,
	                                 ix_ResetEnergySave := FALSE,
	                                 qUDT_HMIStatus => #iqUDT_WorkstationStatus."470".Conveyor,
	                                 qUDT_Status => #iqUDT_WorkstationCommonStatus."470",
	                                 iqUDT_EquipmentControl := #iqUDT_EquipmentControl,
	                                 iqUDT_ConveyorCommand := #iqUDT_WorkstationCommands."470".Conveyor,
	                                 iqUDT_ConveyorInterface := #sUDT_Interface470,
	                                 iqUDT_HandShakeUp := #sUDT_Handshake460,
	                                 iqUDT_HandShake := #sUDT_Handshake470,
	                                 iqUDT_Statistics := #iqUDT_WorkstationStatistics."470".Conveyor);

	            END_REGION
	            REGION MCO

	                #sFB_MCOConveyLinxAixController470(iUDT_AixConfig := #iUDT_Configuration."470".MCO_M01,
	                                                   iUDT_AixInputsModule := #iUDT_MotorInput470,
	                                                   ix_24vOk := #ix_24vOk,
	                                                   ix_SimulationModeActive := "DB_Memory".Simulation,
	                                                   ii_MotorPositionId := 1,
	                                                   qUDT_HMIStatus => #iqUDT_WorkstationStatus."470".MCO_M01,
	                                                   iqUDT_AixOutputsModule := #qUDT_MotorOutput470,
	                                                   iqUDT_ConveyorInterface := #sUDT_Interface470,
	                                                   iqUDT_MCOStatistics := #iqUDT_WorkstationStatistics."470".MCO_M01);
	            END_REGION
	        END_REGION

	        REGION 480

	            REGION Displacement
	                #sFB_Displacement480(#sUDT_Interface480);
	            END_REGION

	            REGION EoS

	                #sFB_PEC480(ix_PEC := #iUDT_MotorInput480.AllSensorPortInputs.LeftSensor,
	                            iUDT_PECConfiguration := #iUDT_Configuration."480".PEC_EoS,
	                            qUDT_HMIStatus => #iqUDT_WorkstationStatus."480".PEC_EoS,
	                            iqUDT_ConveyorInterface := #sUDT_Interface480,
	                            iqUDT_PECStatistics := #iqUDT_WorkstationStatistics."480".PEC_EoS);

	            END_REGION

	            REGION Scanner

	                #sFB_CognexDM480(iUDT_CognexDM260_IN := #iUDT_ScannerInput480,
	                                 iqUDT_EquipmentControl := #iqUDT_EquipmentControl,
	                                 ix_Trigger := NOT #iqUDT_WorkstationStatus."480".PEC_EoS.PEC,
	                                 qUDT_CognexDM260_OUT => #qUDT_ScannerOutput480,
	                                 qs_Barcode => #ss_Barcode480,
	                                 qw_RetVal => #tw_dummy);

	            END_REGION

	            REGION Conveyor

	                #sUDT_Handshake480.RTR := #sUDT_Handshake480.RTR OR #iqUDT_WorkstationStatus."480".PEC_EoS.PEC;

	                #sFB_Conveyor480(iUDT_ConveyorConfiguration := #iUDT_Configuration."480".Conveyor,
	                                 idi_PECEoSDistance := #iUDT_Configuration."480".PEC_EoS.Distance,
	                                 idi_PECBoSDistance := 0,
	                                 ii_ExternalSpeed := 0,
	                                 ix_SafetyOk := #ix_SafetyOk,
	                                 ix_24vOk := #ix_24vOk,
	                                 ix_400vOk := #ix_400vOk,
	                                 ix_HardwareOk := #ix_HardwareOk,
	                                 ix_PECEoS := #iqUDT_WorkstationStatus."480".PEC_EoS.PEC,
	                                 ix_PECBoS := TRUE,
	                                 ix_ReverseDirection := FALSE,
	                                 ix_ExternalRequestDieBack := FALSE,
	                                 ix_ExternalRequestHold := FALSE,
	                                 ix_ResetEnergySave := FALSE,
	                                 qUDT_HMIStatus => #iqUDT_WorkstationStatus."480".Conveyor,
	                                 qUDT_Status => #iqUDT_WorkstationCommonStatus."480",
	                                 iqUDT_EquipmentControl := #iqUDT_EquipmentControl,
	                                 iqUDT_ConveyorCommand := #iqUDT_WorkstationCommands."480".Conveyor,
	                                 iqUDT_ConveyorInterface := #sUDT_Interface480,
	                                 iqUDT_HandShakeUp := #sUDT_Handshake470,
	                                 iqUDT_HandShake := #sUDT_Handshake480,
	                                 iqUDT_Statistics := #iqUDT_WorkstationStatistics."480".Conveyor);

	            END_REGION

	            REGION MCO

	                #sFB_MCOConveyLinxAixController480(iUDT_AixConfig := #iUDT_Configuration."480".MCO_M01,
	                                                   iUDT_AixInputsModule := #iUDT_MotorInput480,
	                                                   ix_24vOk := #ix_24vOk,
	                                                   ix_SimulationModeActive := "DB_Memory".Simulation,
	                                                   ii_MotorPositionId := 1,
	                                                   qUDT_HMIStatus => #iqUDT_WorkstationStatus."480".MCO_M01,
	                                                   iqUDT_AixOutputsModule := #qUDT_MotorOutput480,
	                                                   iqUDT_ConveyorInterface := #sUDT_Interface480,
	                                                   iqUDT_MCOStatistics := #iqUDT_WorkstationStatistics."480".MCO_M01);
	            END_REGION
	        END_REGION


	        REGION 490

	            REGION Displacement
	                #sFB_Displacement490(#sUDT_Interface490);
	            END_REGION

	            REGION MCO

	                #sFB_MCOConveyLinxAixController490(iUDT_AixConfig := #iUDT_Configuration."490".MCO_M01,
	                                                   iUDT_AixInputsModule := #iUDT_MotorInput490,
	                                                   ii_PositionSetpoint := #iqUDT_RATPositioning490.Lower.EndPosition,
	                                                   ix_24vOk := #ix_24vOk,
	                                                   ix_SimulationModeActive := "DB_Memory".Simulation,
	                                                   ii_MotorPositionId := 1,
	                                                   ix_StartPositioning := #iqUDT_RATPositioning490.Lower.Start,
	                                                   ix_ResetPosition := #iqUDT_RATPositioning490.Lower.ResetPosition,
	                                                   qUDT_HMIStatus => #iqUDT_WorkstationStatus."490".MCO_M01,
	                                                   qx_Positioned => #iqUDT_RATPositioning490.Lower.Done,
	                                                   iqUDT_AixOutputsModule := #qUDT_MotorOutput490,
	                                                   iqUDT_ConveyorInterface := #sUDT_Interface490,
	                                                   iqUDT_MCOStatistics := #iqUDT_WorkstationStatistics."490".MCO_M01);
	            END_REGION
	        END_REGION


	        REGION 491

	            REGION Displacement
	                #sFB_Displacement491(#sUDT_Interface491);
	            END_REGION

	            REGION RAT

	                #sFB_RightAngledTransfer491(iUDT_Configuration := #iUDT_Configuration."491".RightAngledTransfer,
	                                            iUDT_LowerConveyorConfiguration := #iUDT_Configuration."490".Conveyor,
	                                            iUDT_UpperConveyorConfiguration := #iUDT_Configuration."491".Conveyor,
	                                            iUDT_PECConfiguration := #iUDT_Configuration."490".PEC_EoS,
	                                            ii_DestinationA := #si_DestinationA491,
	                                            ii_DestinationB := 0,
	                                            ii_DestinationC := 0,
	                                            ii_DestinationD := 0,
	                                            ix_HardwareOk := #ix_HardwareOk,
	                                            ix_400vOk := #ix_400vOk,
	                                            ix_24vOk := #ix_24vOk,
	                                            ix_SafetyOk := #ix_SafetyOk,
	                                            ix_AirPressureOk := #ix_AirPressureOk,
	                                            ix_SectionIsDown := #ix_SectionIsDown491,
	                                            ix_SectionIsUp := #ix_SectionIsUp491,
	                                            ix_ConveyorAAuto := #iqUDT_WorkstationCommonStatus."480".AutoON,
	                                            ix_ConveyorBAuto := FALSE,
	                                            ix_ConveyorCAuto := FALSE,
	                                            ix_ConveyorDAuto := #iqUDT_WorkstationCommonStatus."500".AutoON,
	                                            ix_PEC := #iUDT_MotorInput490.AllSensorPortInputs.LeftSensor,
	                                            ix_ExternalReceiveRequestA := NOT #iqUDT_WorkstationStatus."480".PEC_EoS.PEC,
	                                            ix_ExternalReceiveRequestB := FALSE,
	                                            ix_ExternalReceiveRequestC := FALSE,
	                                            ix_ExternalReceiveRequestD := FALSE,
	                                            ix_PECInfeedA := #iqUDT_WorkstationStatus."480".PEC_EoS.PEC,
	                                            qUDT_HMIRATStatus => #iqUDT_WorkstationStatus."491".RightAngledTransfer,
	                                            qUDT_HMIConveyorStatus => #iqUDT_WorkstationStatus."490".Conveyor,
	                                            qUDT_HMIPECStatus => #iqUDT_WorkstationStatus."491".PEC_EoS,
	                                            qUDT_RATStatus => #iqUDT_WorkstationCommonStatus."491",
	                                            qUDT_ConveyorStatus => #iqUDT_WorkstationCommonStatus."490",
	                                            qx_PopupControl => #qx_PopupControl491,
	                                            qx_ExternalSendRequestA => #tx_dummy,
	                                            qx_ExternalSendRequestB => #tx_dummy,
	                                            qx_ExternalSendRequestC => #tx_dummy,
	                                            qx_ExternalSendRequestD => #tx_dummy,
	                                            iqUDT_EquipmentControl := #iqUDT_EquipmentControl,
	                                            iqUDT_RATCommand := #iqUDT_WorkstationCommands."491".RAT,
	                                            iqUDT_ConveyorCommand := #iqUDT_WorkstationCommands."490".Conveyor,
	                                            iqUDT_RATStatistics := #iqUDT_WorkstationStatistics."491".RightAngledTransfer,
	                                            iqUDT_ConveyorStatistics := #iqUDT_WorkstationStatistics."490".Conveyor,
	                                            iqUDT_PECStatistics := #iqUDT_WorkstationStatistics."491".PEC_EoS,
	                                            iqUDT_HandShakeConveyorA := #sUDT_Handshake480,
	                                            iqUDT_HandShakeConveyorB := #tUDT_dummyHandshake,
	                                            iqUDT_HandShakeConveyorC := #tUDT_dummyHandshake,
	                                            iqUDT_HandShakeConveyorD := #sUDT_Handshake491,
	                                            iqUDT_LowerConveyorInterface := #sUDT_Interface490,
	                                            iqUDT_UpperConveyorInterface := #sUDT_Interface491,
	                                            iqUDT_RATPositioning := #iqUDT_RATPositioning490,
	                                            iqUDT_BladeStopEoSInterface := #tUDT_DummyBladeStop,
	                                            iqUDT_BladeStopBoSInterface := #tUDT_DummyBladeStop);



	            END_REGION

	            REGION MCO

	                #sFB_MCOConveyLinxAixController491(iUDT_AixConfig := #iUDT_Configuration."491".MCO_M01,
	                                                   iUDT_AixInputsModule := #iUDT_MotorInput490,
	                                                   ix_24vOk := #ix_24vOk,
	                                                   ix_SimulationModeActive := "DB_Memory".Simulation,
	                                                   ii_MotorPositionId := 2,
	                                                   qUDT_HMIStatus => #iqUDT_WorkstationStatus."491".MCO_M01,
	                                                   iqUDT_AixOutputsModule := #qUDT_MotorOutput490,
	                                                   iqUDT_ConveyorInterface := #sUDT_Interface491,
	                                                   iqUDT_MCOStatistics := #iqUDT_WorkstationStatistics."491".MCO_M01);
	            END_REGION

	        END_REGION

	        REGION 500

	            REGION Displacement
	                #sFB_Displacement500(#sUDT_Interface500);
	            END_REGION

	            REGION EoS

	                #sFB_PEC500(ix_PEC := #iUDT_MotorInput500.AllSensorPortInputs.LeftSensor,
	                            iUDT_PECConfiguration := #iUDT_Configuration."500".PEC_EoS,
	                            qUDT_HMIStatus => #iqUDT_WorkstationStatus."500".PEC_EoS,
	                            iqUDT_ConveyorInterface := #sUDT_Interface500,
	                            iqUDT_PECStatistics := #iqUDT_WorkstationStatistics."500".PEC_EoS);

	            END_REGION
	            REGION Conveyor

	                #sUDT_Handshake500.RTR := #sUDT_Handshake500.RTR OR #iqUDT_WorkstationStatus."500".PEC_EoS.PEC;

	                #sFB_Conveyor500(iUDT_ConveyorConfiguration := #iUDT_Configuration."500".Conveyor,
	                                 idi_PECEoSDistance := #iUDT_Configuration."500".PEC_EoS.Distance,
	                                 idi_PECBoSDistance := 0,
	                                 ii_ExternalSpeed := 0,
	                                 ix_SafetyOk := #ix_SafetyOk,
	                                 ix_24vOk := #ix_24vOk,
	                                 ix_400vOk := #ix_400vOk,
	                                 ix_HardwareOk := #ix_HardwareOk,
	                                 ix_PECEoS := #iqUDT_WorkstationStatus."500".PEC_EoS.PEC,
	                                 ix_PECBoS := TRUE,
	                                 ix_ReverseDirection := FALSE,
	                                 ix_ExternalRequestDieBack := FALSE,
	                                 ix_ExternalRequestHold := FALSE,
	                                 ix_ResetEnergySave := FALSE,
	                                 qUDT_HMIStatus => #iqUDT_WorkstationStatus."500".Conveyor,
	                                 qUDT_Status => #iqUDT_WorkstationCommonStatus."500",
	                                 iqUDT_EquipmentControl := #iqUDT_EquipmentControl,
	                                 iqUDT_ConveyorCommand := #iqUDT_WorkstationCommands."500".Conveyor,
	                                 iqUDT_ConveyorInterface := #sUDT_Interface500,
	                                 iqUDT_HandShakeUp := #sUDT_Handshake491,
	                                 iqUDT_HandShake := #sUDT_Handshake500,
	                                 iqUDT_Statistics := #iqUDT_WorkstationStatistics."500".Conveyor);

	            END_REGION
	            REGION MCO

	                #sFB_MCOConveyLinxAixController500(iUDT_AixConfig := #iUDT_Configuration."500".MCO_M01,
	                                                   iUDT_AixInputsModule := #iUDT_MotorInput500,
	                                                   ix_24vOk := #ix_24vOk,
	                                                   ix_SimulationModeActive := "DB_Memory".Simulation,
	                                                   ii_MotorPositionId := 1,
	                                                   qUDT_HMIStatus => #iqUDT_WorkstationStatus."500".MCO_M01,
	                                                   iqUDT_AixOutputsModule := #qUDT_MotorOutput500,
	                                                   iqUDT_ConveyorInterface := #sUDT_Interface500,
	                                                   iqUDT_MCOStatistics := #iqUDT_WorkstationStatistics."500".MCO_M01);
	            END_REGION
	        END_REGION
	    END_IF;
	END_REGION

	REGION 6 - Station Outfeed
	    REGION 610

	        REGION Displacement
	            #sFB_Displacement610(#sUDT_Interface610);
	        END_REGION

	        REGION MCO

	            #sFB_MCOConveyLinxAixController610(iUDT_AixConfig := #iUDT_Configuration."610".MCO_M01,
	                                               iUDT_AixInputsModule := #iUDT_MotorInput610,
	                                               ix_24vOk := #ix_24vOk,
	                                               ix_SimulationModeActive := "DB_Memory".Simulation,
	                                               ii_MotorPositionId := 1,
	                                               qUDT_HMIStatus => #iqUDT_WorkstationStatus."610".MCO_M01,
	                                               iqUDT_AixOutputsModule := #qUDT_MotorOutput610,
	                                               iqUDT_ConveyorInterface := #sUDT_Interface610,
	                                               iqUDT_MCOStatistics := #iqUDT_WorkstationStatistics."610".MCO_M01);
	        END_REGION
	    END_REGION

	    REGION 611

	        REGION Displacement
	            #sFB_Displacement611(#sUDT_Interface611);
	        END_REGION

	        REGION RAT

	            #sFB_RightAngledTransfer611(iUDT_Configuration := #iUDT_Configuration."611".RightAngledTransfer,
	                                        iUDT_LowerConveyorConfiguration := #iUDT_Configuration."610".Conveyor,
	                                        iUDT_UpperConveyorConfiguration := #iUDT_Configuration."611".Conveyor,
	                                        iUDT_PECConfiguration := #iUDT_Configuration."610".PEC_EoS,
	                                        ii_DestinationA := 0,
	                                        ii_DestinationB := 0,
	                                        ii_DestinationC := 1,
	                                        ii_DestinationD := 1,
	                                        ix_HardwareOk := #ix_HardwareOk,
	                                        ix_400vOk := #ix_400vOk,
	                                        ix_24vOk := #ix_24vOk,
	                                        ix_SafetyOk := #ix_SafetyOk,
	                                        ix_AirPressureOk := #ix_AirPressureOk,
	                                        ix_SectionIsDown := #ix_SectionIsDown611,
	                                        ix_SectionIsUp := #ix_SectionIsUp611,
	                                        ix_ConveyorAAuto := TRUE,
	                                        ix_ConveyorBAuto := #iqUDT_WorkstationCommonStatus."620".AutoON,
	                                        ix_ConveyorCAuto := #iqUDT_WorkstationCommonStatus."500".AutoON,
	                                        ix_ConveyorDAuto := #iqUDT_WorkstationCommonStatus."300".AutoON,
	                                        ix_PEC := #iUDT_MotorInput610.AllSensorPortInputs.LeftSensor,
	                                        ix_ExternalReceiveRequestA := FALSE,
	                                        ix_ExternalReceiveRequestB := FALSE,
	                                        ix_ExternalReceiveRequestC := NOT #iqUDT_WorkstationStatus."500".PEC_EoS.PEC,
	                                        ix_ExternalReceiveRequestD := NOT #iqUDT_WorkstationStatus."300".PEC_EoS.PEC,
	                                        ix_PECInfeedC := #iqUDT_WorkstationStatus."500".PEC_EoS.PEC,
	                                        ix_PECInfeedD := #iqUDT_WorkstationStatus."300".PEC_EoS.PEC,
	                                        qUDT_HMIRATStatus => #iqUDT_WorkstationStatus."611".RightAngledTransfer,
	                                        qUDT_HMIConveyorStatus => #iqUDT_WorkstationStatus."610".Conveyor,
	                                        qUDT_HMIPECStatus => #iqUDT_WorkstationStatus."611".PEC_EoS,
	                                        qUDT_RATStatus => #iqUDT_WorkstationCommonStatus."611",
	                                        qUDT_ConveyorStatus => #iqUDT_WorkstationCommonStatus."610",
	                                        qx_PopupControl => #qx_PopupControl611,
	                                        qx_ExternalSendRequestA => #tx_dummy,
	                                        qx_ExternalSendRequestB => #tx_dummy,
	                                        qx_ExternalSendRequestC => #tx_dummy,
	                                        qx_ExternalSendRequestD => #tx_dummy,
	                                        iqUDT_EquipmentControl := #iqUDT_EquipmentControl,
	                                        iqUDT_RATCommand := #iqUDT_WorkstationCommands."611".RightAngledTransfer,
	                                        iqUDT_ConveyorCommand := #iqUDT_WorkstationCommands."610".Conveyor,
	                                        iqUDT_RATStatistics := #iqUDT_WorkstationStatistics."611".RightAngledTransfer,
	                                        iqUDT_ConveyorStatistics := #iqUDT_WorkstationStatistics."610".Conveyor,
	                                        iqUDT_PECStatistics := #iqUDT_WorkstationStatistics."611".PEC_EoS,
	                                        iqUDT_HandShakeConveyorA := #tUDT_dummyHandshake,
	                                        iqUDT_HandShakeConveyorB := #sUDT_Handshake610,
	                                        iqUDT_HandShakeConveyorC := #sUDT_Handshake500,
	                                        iqUDT_HandShakeConveyorD := #sUDT_Handshake300,
	                                        iqUDT_LowerConveyorInterface := #sUDT_Interface610,
	                                        iqUDT_UpperConveyorInterface := #sUDT_Interface611,
	                                        iqUDT_RATPositioning := #iqUDT_RATPositioning610,
	                                        iqUDT_BladeStopEoSInterface := #tUDT_DummyBladeStop,
	                                        iqUDT_BladeStopBoSInterface := #tUDT_DummyBladeStop);



	        END_REGION

	        REGION MCO

	            #sFB_MCOConveyLinxAixController611(iUDT_AixConfig := #iUDT_Configuration."611".MCO_M01,
	                                               iUDT_AixInputsModule := #iUDT_MotorInput610,
	                                               ii_PositionSetpoint := #iqUDT_RATPositioning610.Upper.EndPosition,
	                                               ix_24vOk := #ix_24vOk,
	                                               ix_SimulationModeActive := "DB_Memory".Simulation,
	                                               ii_MotorPositionId := 2,
	                                               ix_StartPositioning := #iqUDT_RATPositioning610.Upper.Start,
	                                               ix_ResetPosition := #iqUDT_RATPositioning610.Upper.ResetPosition,
	                                               qUDT_HMIStatus => #iqUDT_WorkstationStatus."611".MCO_M01,
	                                               qx_Positioned => #iqUDT_RATPositioning610.Upper.Done,
	                                               iqUDT_AixOutputsModule := #qUDT_MotorOutput610,
	                                               iqUDT_ConveyorInterface := #sUDT_Interface611,
	                                               iqUDT_MCOStatistics := #iqUDT_WorkstationStatistics."611".MCO_M01);
	        END_REGION

	    END_REGION

	    REGION 620

	        REGION Displacement
	            #sFB_Displacement620(#sUDT_Interface620);
	        END_REGION

	        REGION Conveyor

	            #sFB_Conveyor620(iUDT_ConveyorConfiguration := #iUDT_Configuration."620".Conveyor,
	                             idi_PECEoSDistance := 0,
	                             idi_PECBoSDistance := 0,
	                             ii_ExternalSpeed := 0,
	                             ix_SafetyOk := #ix_SafetyOk,
	                             ix_24vOk := #ix_24vOk,
	                             ix_400vOk := #ix_400vOk,
	                             ix_HardwareOk := #ix_HardwareOk,
	                             ix_PECEoS := TRUE,
	                             ix_PECBoS := TRUE,
	                             ix_ReverseDirection := FALSE,
	                             ix_ExternalRequestDieBack := FALSE,
	                             ix_ExternalRequestHold := FALSE,
	                             ix_ResetEnergySave := FALSE,
	                             qUDT_HMIStatus => #iqUDT_WorkstationStatus."620".Conveyor,
	                             qUDT_Status => #iqUDT_WorkstationCommonStatus."620",
	                             iqUDT_EquipmentControl := #iqUDT_EquipmentControl,
	                             iqUDT_ConveyorCommand := #iqUDT_WorkstationCommands."620".Conveyor,
	                             iqUDT_ConveyorInterface := #sUDT_Interface620,
	                             iqUDT_HandShakeUp := #sUDT_Handshake610,
	                             iqUDT_HandShake := #sUDT_Handshake620,
	                             iqUDT_Statistics := #iqUDT_WorkstationStatistics."620".Conveyor);

	        END_REGION

	        REGION MCO

	            #sFB_MCOConveyLinxAixController620(iUDT_AixConfig := #iUDT_Configuration."620".MCO_M01,
	                                               iUDT_AixInputsModule := #iUDT_MotorInput620,
	                                               ix_24vOk := #ix_24vOk,
	                                               ix_SimulationModeActive := "DB_Memory".Simulation,
	                                               ii_MotorPositionId := 1,
	                                               qUDT_HMIStatus => #iqUDT_WorkstationStatus."620".MCO_M01,
	                                               iqUDT_AixOutputsModule := #qUDT_MotorOutput620,
	                                               iqUDT_ConveyorInterface := #sUDT_Interface620,
	                                               iqUDT_MCOStatistics := #iqUDT_WorkstationStatistics."620".MCO_M01);
	        END_REGION

	    END_REGION

	    REGION 630

	        REGION Displacement
	            #sFB_Displacement630(#sUDT_Interface630);
	        END_REGION

	        REGION Conveyor

	            #sFB_Conveyor630(iUDT_ConveyorConfiguration := #iUDT_Configuration."630".Conveyor,
	                             idi_PECEoSDistance := 0,
	                             idi_PECBoSDistance := 0,
	                             ii_ExternalSpeed := 0,
	                             ix_SafetyOk := #ix_SafetyOk,
	                             ix_24vOk := #ix_24vOk,
	                             ix_400vOk := #ix_400vOk,
	                             ix_HardwareOk := #ix_HardwareOk,
	                             ix_PECEoS := TRUE,
	                             ix_PECBoS := TRUE,
	                             ix_ReverseDirection := FALSE,
	                             ix_ExternalRequestDieBack := FALSE,
	                             ix_ExternalRequestHold := FALSE,
	                             ix_ResetEnergySave := FALSE,
	                             qUDT_HMIStatus => #iqUDT_WorkstationStatus."630".Conveyor,
	                             qUDT_Status => #iqUDT_WorkstationCommonStatus."630",
	                             iqUDT_EquipmentControl := #iqUDT_EquipmentControl,
	                             iqUDT_ConveyorCommand := #iqUDT_WorkstationCommands."630".Conveyor,
	                             iqUDT_ConveyorInterface := #sUDT_Interface630,
	                             iqUDT_HandShakeUp := #sUDT_Handshake620,
	                             iqUDT_HandShake := #sUDT_Handshake630,
	                             iqUDT_Statistics := #iqUDT_WorkstationStatistics."630".Conveyor);

	        END_REGION

	        REGION MCO

	            #sFB_MCOConveyLinxAixController630(iUDT_AixConfig := #iUDT_Configuration."630".MCO_M01,
	                                               iUDT_AixInputsModule := #iUDT_MotorInput630,
	                                               ix_24vOk := #ix_24vOk,
	                                               ix_SimulationModeActive := "DB_Memory".Simulation,
	                                               ii_MotorPositionId := 1,
	                                               qUDT_HMIStatus => #iqUDT_WorkstationStatus."630".MCO_M01,
	                                               iqUDT_AixOutputsModule := #qUDT_MotorOutput630,
	                                               iqUDT_ConveyorInterface := #sUDT_Interface630,
	                                               iqUDT_MCOStatistics := #iqUDT_WorkstationStatistics."630".MCO_M01);
	        END_REGION
	    END_REGION

	    REGION 640

	        REGION Displacement
	            #sFB_Displacement640(#sUDT_Interface640);
	        END_REGION

	        REGION EoS

	            #sFB_PEC640(ix_PEC := #iUDT_MotorInput640.AllSensorPortInputs.LeftSensor,
	                        iUDT_PECConfiguration := #iUDT_Configuration."640".PEC_EoS,
	                        qUDT_HMIStatus => #iqUDT_WorkstationStatus."640".PEC_EoS,
	                        iqUDT_ConveyorInterface := #sUDT_Interface640,
	                        iqUDT_PECStatistics := #iqUDT_WorkstationStatistics."640".PEC_EoS);

	        END_REGION
	        REGION Conveyor

	            #sFB_Conveyor640(iUDT_ConveyorConfiguration := #iUDT_Configuration."640".Conveyor,
	                             idi_PECEoSDistance := #iUDT_Configuration."640".PEC_EoS.Distance,
	                             idi_PECBoSDistance := 0,
	                             ii_ExternalSpeed := 0,
	                             ix_SafetyOk := #ix_SafetyOk,
	                             ix_24vOk := #ix_24vOk,
	                             ix_400vOk := #ix_400vOk,
	                             ix_HardwareOk := #ix_HardwareOk,
	                             ix_PECEoS := #iqUDT_WorkstationStatus."640".PEC_EoS.PEC,
	                             ix_PECBoS := TRUE,
	                             ix_ReverseDirection := FALSE,
	                             ix_ExternalRequestDieBack := FALSE,
	                             ix_ExternalRequestHold := FALSE,
	                             ix_ResetEnergySave := FALSE,
	                             qUDT_HMIStatus => #iqUDT_WorkstationStatus."640".Conveyor,
	                             qUDT_Status => #iqUDT_WorkstationCommonStatus."640",
	                             iqUDT_EquipmentControl := #iqUDT_EquipmentControl,
	                             iqUDT_ConveyorCommand := #iqUDT_WorkstationCommands."640".Conveyor,
	                             iqUDT_ConveyorInterface := #sUDT_Interface640,
	                             iqUDT_HandShakeUp := #sUDT_Handshake630,
	                             iqUDT_HandShake := #iqUDT_HandshakeDownstream640,
	                             iqUDT_Statistics := #iqUDT_WorkstationStatistics."640".Conveyor);

	        END_REGION

	        REGION MCO

	            #sFB_MCOConveyLinxAixController640(iUDT_AixConfig := #iUDT_Configuration."640".MCO_M01,
	                                               iUDT_AixInputsModule := #iUDT_MotorInput640,
	                                               ix_24vOk := #ix_24vOk,
	                                               ix_SimulationModeActive := "DB_Memory".Simulation,
	                                               ii_MotorPositionId := 1,
	                                               qUDT_HMIStatus => #iqUDT_WorkstationStatus."640".MCO_M01,
	                                               iqUDT_AixOutputsModule := #qUDT_MotorOutput640,
	                                               iqUDT_ConveyorInterface := #sUDT_Interface640,
	                                               iqUDT_MCOStatistics := #iqUDT_WorkstationStatistics."640".MCO_M01);
	        END_REGION
	    END_REGION
	END_REGION


END_FUNCTION_BLOCK

FUNCTION_BLOCK "FB_CaptureRATPosition"
TITLE = Capturing RAT position when product leave infeed belt
{ S7_Optimized_Access := 'TRUE' }
AUTHOR : 'Kamil Pokorski'
VERSION : 1.0
// ATTRIBUTES
// AUTO_NUMBER = True
// BLOCK_NUMBER = 260
// END_ATTRIBUTES
//This block should be used only in Cyclic interrupt. All connected IO must be periferal.
   VAR_INPUT
      ix_InfeedPEC { ExternalAccessible := 'False'; ExternalVisible := 'False'; ExternalWritable := 'False'} : Bool;   // TRUE when RAT infeed PEC is clear
      ix_Request { ExternalAccessible := 'False'; ExternalVisible := 'False'; ExternalWritable := 'False'} : Bool;
      ii_MotorPosition { ExternalAccessible := 'False'; ExternalVisible := 'False'; ExternalWritable := 'False'} : Int;   // RAT motor position (lower when infeeding on lower position, upper if infeeding on upper position)
   END_VAR

   VAR_IN_OUT
      iqi_Position { ExternalAccessible := 'False'; ExternalVisible := 'False'; ExternalWritable := 'False'} : Int;   // Captured position
   END_VAR

   VAR
      sR_TRIG_InfeedPEC {InstructionName := 'R_TRIG'; LibVersion := '1.0'; ExternalAccessible := 'False'; ExternalVisible := 'False'; ExternalWritable := 'False'; S7_SetPoint := 'False'} : R_TRIG;   // Detecting rising edge on infeed PEC
   END_VAR


BEGIN
	(*
	----------------------------------------------------------------------------------------

	Version history:
	Date        | Version   | Author        | Remark
	----------------------------------------------------------------------------------------
	27/05/2024  | 1.0       | K.Pokorski    | Initial version
	*)

	#sR_TRIG_InfeedPEC(CLK := #ix_InfeedPEC);

	IF #sR_TRIG_InfeedPEC.Q AND #ix_Request THEN
	    #iqi_Position := #ii_MotorPosition;
	END_IF;


END_FUNCTION_BLOCK

